Yaskawa INFORM job: CUT_ONLY.JBI

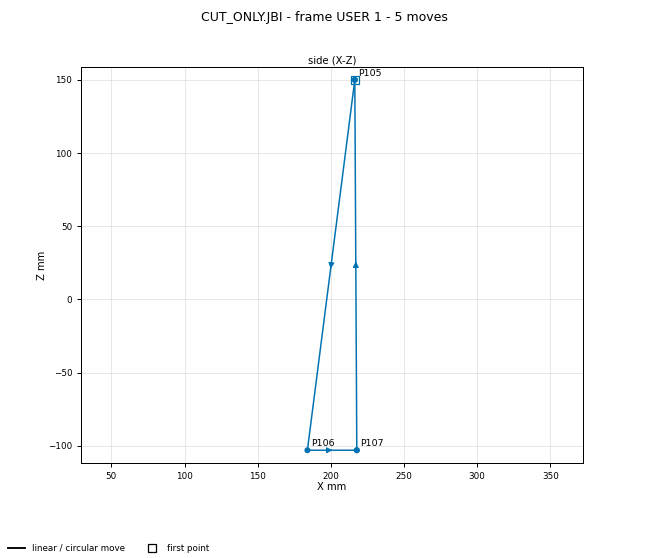
[picture p0: tool path of CUT_ONLY.JBI in frame USER 1, 5 of 7 moves have a stored position in this frame; points joined in program order, loops and branches not executed]
/JOB
//NAME CUT_ONLY
//POS
///NPOS 0,0,0,6,0,0
///TOOL 0
///POSTYPE BASE
///RECTAN
///RCONF 1,0,0,0,0,0,0,0,0,0,0,0,0,0,0,0,0,0,0,0,0,0,0,0
P00100=275.000,0.000,875.000,180.0000,45.0000,0.0000
///USER 1
///POSTYPE USER
P00105=216.374,-55.365,150.000,179.9941,-0.0013,-179.9943
P00106=183.974,-55.386,-103.111,179.9969,-0.0014,-179.9945
P00107=217.725,-55.392,-103.109,179.9979,-0.0019,-179.9959
P00108=217.733,-59.426,-103.121,179.9979,-0.0009,-179.9957
P00109=216.373,-55.365,149.996,179.9952,-0.0016,-179.9953
//INST
///DATE 2023/01/24 16:29
///ATTR SC,RW
///GROUP1 RB1
NOP
MOVJ P100 VJ=50.00
'CUT*****************************
MOVJ P105 VJ=25.00  //APPROCH CUT
MOVL P106 V=150.0 PL=0  //CUT PRE-SLIDE
MOVL P107 V=150.0 PL=0  //CUT SLIDE
MOVL P108 V=150.0 PL=0  //CUT TOUCH
' Inch welding wire
PULSE OT#(3003) T=0.50
TIMER T=0.50
PULSE OT#(2819) T=1.00
TIMER T=1.00
MOVL P109 V=150.0  //DEPART CUT
'********************************
MOVJ P100 VJ=50.00
END
